TYPE Uuid : STRING; END_TYPE

(* stored: Version 1.1.0.1, ProductVersion 3.1.4024.12
   DUT Uuid: Id {9bed3ba9-dce5-0c02-2327-56295ac00212} *)
